Staubli VAL3: onEdit.pgx

public program onEdit(string& x_sItem[])
  local string l_sItem[3]
  local num l_nCount
  local string l_sFlag[3]
  local string l_sName[3]
  local num i
  local string l_sData
  local num l_nFlag
  local string l_sMessage
  local num l_nNum
  local string l_sId
begin
  // show the real name
  l_sData=x_sItem
  do
    // sMode
    i=find(l_sData,"AND")
    if i!=-1
      i=i+len("AND")+1
    else
      i=find(l_sData,"OR")
      if i!=-1
        i=i+len("OR")+1
      endIf
    endIf
    //
    if i!=-1
      l_sItem[l_nCount]=left(l_sData,i)
      l_sData=right(l_sData,len(l_sData)-i)
    else
      l_sItem[l_nCount]=l_sData
    endIf
    l_nFlag=find(l_sItem[l_nCount],">")
    // l_bMode
    if find(l_sItem[l_nCount],">ON")!=-1
      l_sFlag[l_nCount]=">ON"+chr(10)
    else
      l_sFlag[l_nCount]=">OFF"+chr(10)
    endIf
    // sItem
    l_sItem[l_nCount]=left(l_sItem[l_nCount],l_nFlag)
    l_sId=l_sItem[l_nCount]
    l_sName[l_nCount]=saveInOut:dInput[l_sId].sName
    l_nCount=l_nCount+1
  until i==-1
  // show the ID+name
  l_sMessage=""
  for i=0 to 2
    if l_sItem[i]!=""
      l_sMessage=l_sMessage+l_sItem[i]+"["+l_sName[i]+"]"+l_sFlag[i]
    endIf
  endFor
  // popUp IT
  popUpMsg(l_sMessage)
end
